{attribute 'linkalways'} 
{attribute 'no_explicit_call' := 'This FB is a CLASS and must be accessed using methods or properties'}
{attribute 'enable_dynamic_creation'}
FUNCTION_BLOCK FINAL MAX_DINT EXTENDS Node
VAR
	in1 : _DINT(0);
	in2 : _DINT(0);
	out : _DINT(0);
END_VAR

METHOD PUBLIC Clone : I_Node
VAR
	pNode : POINTER TO MAX_DINT;
END_VAR
pNode := __NEW(MAX_DINT);
Clone := pNode^;
END_METHOD

METHOD FB_init : BOOL
VAR_INPUT
	bInitRetains : BOOL; // if TRUE, the retain variables are initialized (warm start / cold start)
	bInCopyCode : BOOL;  // if TRUE, the instance afterwards gets moved into the copy code (online change)
END_VAR
AddInput('in1',THIS^.in1);
AddInput('in2',THIS^.in2);
AddOutput('out', THIS^.out);
END_METHOD

METHOD PROTECTED OnExecute
VAR
END_VAR
out.Value := MAX(in1.Value, in2.Value);
END_METHOD

END_FUNCTION_BLOCK

(* stored: Version 1.1.0.1, ProductVersion 3.1.4024.15
   POU MAX_DINT: Id {5a2cf0c0-6605-4da1-9252-a55b0c81ec41}, SpecialFunc None
   Folder Constructor: Id {761b7ee9-4db4-40c4-ac5d-39d97827ec98}
   Method Clone: Id {38454b99-5d9f-4939-a029-fd92215a6a35}
   Method FB_init: Id {f81ee9ed-a7d8-4507-8d64-d2e949e93681}
   Method OnExecute: Id {e8b18fd8-f8d5-432e-841e-1b834be8f0ca} *)
